FUNCTION_BLOCK FB_Base_Test EXTENDS FB_Base
VAR_INPUT
END_VAR
VAR_OUTPUT
END_VAR
VAR
END_VAR

SUPER^(refFbFault := refFbFault);

END_FUNCTION_BLOCK

(* stored: Version 1.1.0.1, ProductVersion 3.1.4024.11
   POU FB_Base_Test: Id {404222a2-3ad1-0183-220a-0115e1efb234}, SpecialFunc None *)
